{attribute 'GeneratedUsingTerminal: EJ7334-0008-0016'}
{attribute addProperty BoxType "EJ7334-0008-0016"}
{attribute addProperty Id "ControlAT %Q*Control_FF5AB9B22VelocityAT %Q*INT2"}
{attribute addProperty CRC "4152316366"}
{attribute addProperty Size "4"}
TYPE DCM_Outputs_Channel_F77F51CE EXTENDS OutputBase_10CEE7DE :
STRUCT
	{attribute addProperty Name "Control"}
	Control AT %Q* : Control_FF5AB9B2;
	{attribute addProperty Name "Velocity"}
	Velocity AT %Q* : INT;
END_STRUCT
END_TYPE

(* stored: Version 1.2.0.0, ProductVersion 3.1.4024.9
   DUT DCM_Outputs_Channel_F77F51CE: Id {e24bb3d5-43d3-4c66-8c32-e4f257e760d6} *)
